PROGRAM MAIN
VAR
	//cmt 1
	bTest_1 :BOOL;
	//cmt 2
	bTest_2 :BOOL;
END_VAR

END_PROGRAM

(* stored: Version 1.1.0.1, ProductVersion 3.1.4024.12
   POU MAIN: Id {551d6576-c260-4cbc-87c2-99b82bf64971}, SpecialFunc None *)
